TYPE HMI_MAN_TemplateMachinePart :
STRUCT
	Cil_Example: HMI_MAN_Valve;
	VCG_Suckers: HMI_MAN_VacuumGenerator;
	Mtr_Example: HMI_MAN_Motor;
	Fdr_Example: HMI_MAN_FDR_CTC300;
	Srv_Example: HMI_MAN_Servo;
	Gantry_Example: HMI_MAN_SingleBeltGantry;
	SrvGripper_Example: HMI_MAN_SRV_GEH6000;
	Cam_OmronSmartCam: HMI_MAN_OmronMicroScan;
	Cam_OmronController: HMI_MAN_OmronCamera;
END_STRUCT
END_TYPE

(* stored: Version 1.1.0.1, ProductVersion 3.1.4024.12
   DUT HMI_MAN_TemplateMachinePart: Id {811c2c62-376c-4b21-b642-8a80912fe820} *)
